(* PLC project  *)

CONFIGURATION Empty_Module_22
END_CONFIGURATION
